{attribute 'TcGenerated'}
// This function has been automatically generated from the project information.
VAR_GLOBAL CONSTANT
	{attribute 'const_non_replaced'}
	{attribute 'linkalways'}
	stLibVersion_OscatBasic : ST_LibVersion := (iMajor := 1, iMinor := 0, iBuild := 0, iRevision := 0, sVersion := '1.0.0');
END_VAR

(* stored: Version 1.1.0.1, ProductVersion 3.1.4022.7
   GVL Global_Version: Id {8cd9474f-8215-4789-93e6-7d64c7a11e0c} *)
